(* CoDeSys 2.3.9.37 project: Cap6_3.pro *)
(* Libraries: Standard.lib 4.10.05 12:14:46 *)

(* POU PLC_PRG, LD *)
PROGRAM PLC_PRG
VAR
	A: BOOL;
   	S1: BOOL;
 	MiTempo: TON;
END_VAR
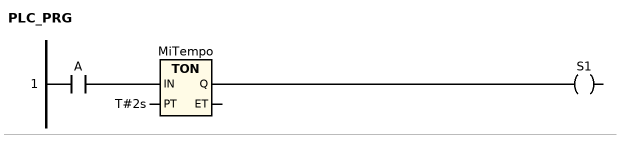
_LD_ (* Ladder Diagram *)
NETWORK 1
	[A] - MiTempo:TON(IN: *, PT: T#2s) --- (S1)
_END_LD_
(* the same logic as Structured Text *)
(* Network 1 *)
MiTempo(IN := A, PT := T#2s);
S1 := MiTempo.Q;
END_PROGRAM

(* Visualisation Visu
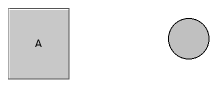
button at (100,80)-(161,151): text "A"; toggles PLC_PRG.A
ellipse at (260,90)-(301,131): alarm colour if PLC_PRG.S1
1 elements of other kinds (tables, trends, ...) not read
*)
